FUNCTION_BLOCK INSTRUCTION_EXTRACTOR (* Composite Function Block Type *)
  (* Standard: 61499-2 *)
  (* Version 0.0, 12/28/2022, Dmitrii, Flexbridge AB, template *)
  PACKAGE UAO.Hackathon;
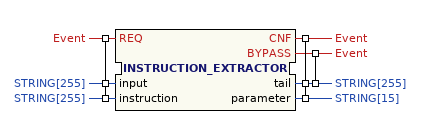
  EVENT_INPUT
    REQ WITH instruction, input; (* Normal Execution Request *)
  END_EVENT
  EVENT_OUTPUT
    CNF WITH tail, parameter; (* Requested instruction found and parsed *)
    BYPASS WITH tail; (* Instruction not found *)
  END_EVENT
  VAR_INPUT
    input : STRING[255]; (* Input string *)
    instruction : STRING[255]; (* Instruction to search for *)
  END_VAR
  VAR_OUTPUT
    tail : STRING[255]; (* Remaining 'tail' of the input string if instruction found, or the whole input string if not. *)
    parameter : STRING[15]; (* Instruction parameter *)
  END_VAR
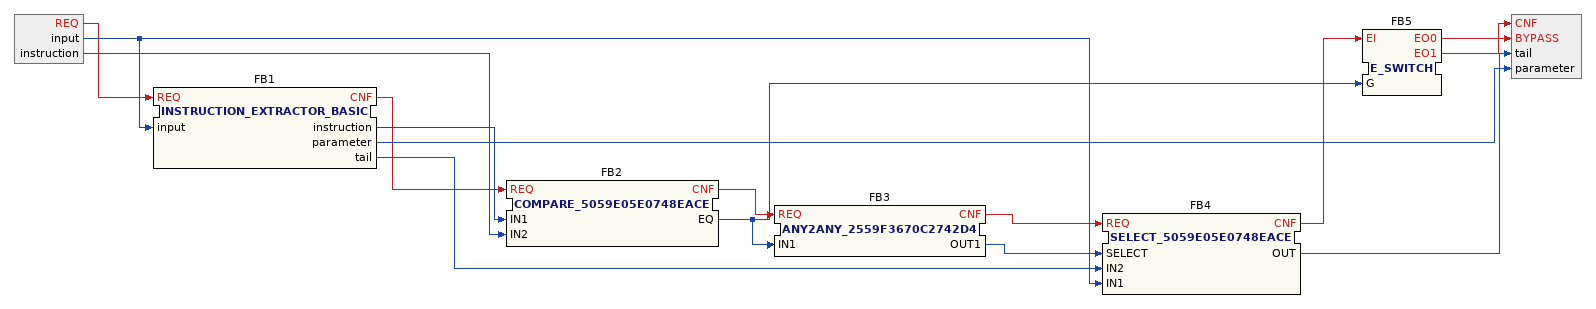
  FBS
    FB1 : INSTRUCTION_EXTRACTOR_BASIC;
    FB2 : COMPARE_5059E05E0748EACE; {SET_ATTRIBUTE(Configuration.GenericFBType.InterfaceParams, Runtime.Standard#CNT:=2;IN${CNT$}:STRING(255))}
    FB4 : SELECT_5059E05E0748EACE; {SET_ATTRIBUTE(Configuration.GenericFBType.InterfaceParams, Runtime.Standard#CNT:=2;IN${CNT$}:STRING(255))}
    FB3 : ANY2ANY_2559F3670C2742D4; {SET_ATTRIBUTE(Configuration.GenericFBType.InterfaceParams, Runtime.Standard#CNT:=1;IN${CNT$}:BOOL;OUT${CNT$}:USINT)}
    FB5 : E_SWITCH;
  END_FBS
  EVENT_CONNECTIONS
    REQ TO FB1.REQ;
    FB3.CNF TO FB4.REQ;
    FB1.CNF TO FB2.REQ;
    FB2.CNF TO FB3.REQ;
    FB4.CNF TO FB5.EI;
    FB5.EO0 TO BYPASS;
    FB5.EO1 TO CNF;
  END_CONNECTIONS
  DATA_CONNECTIONS
    input TO FB1.input;
    FB3.OUT1 TO FB4.SELECT;
    FB1.tail TO FB4.IN2;
    FB4.OUT TO tail;
    FB1.instruction TO FB2.IN1;
    instruction TO FB2.IN2;
    FB2.EQ TO FB3.IN1;
    FB1.parameter TO parameter;
    FB2.EQ TO FB5.G;
    input TO FB4.IN1;
  END_CONNECTIONS
END_FUNCTION_BLOCK
